(* IEC 61131-3 sources: plc-agent/examples, 6 files *)

(* ---- invalid.st ---- *)
PROGRAM Main
VAR_OUTPUT
    Motor : BOOL;
END_VAR

Motor := ;
END_PROGRAM

(* ---- minimal.st ---- *)
PROGRAM Main
VAR_INPUT
    Start : BOOL;
END_VAR
VAR_OUTPUT
    Motor : BOOL;
END_VAR

Motor := Start;
END_PROGRAM

(* ---- motor_start_stop.st ---- *)
PROGRAM Main
VAR
    Start AT %IX0.0 : BOOL;
    Stop AT %IX0.1 : BOOL;
    Motor AT %QX0.0 : BOOL;
END_VAR
VAR
    StartEdge : R_TRIG;
    RunTimer : TON;
    Running : BOOL := FALSE;
END_VAR

StartEdge(CLK := Start);
IF Stop THEN
    Running := FALSE;
ELSIF StartEdge.Q AND NOT Running THEN
    Running := TRUE;
END_IF;

RunTimer(IN := Running, PT := T#10s);
IF RunTimer.Q THEN
    Running := FALSE;
END_IF;
Motor := Running;
END_PROGRAM

CONFIGURATION Config0
    RESOURCE Res0 ON PLC
        TASK MainTask(INTERVAL := T#20ms, PRIORITY := 0);
        PROGRAM Inst0 WITH MainTask : Main;
    END_RESOURCE
END_CONFIGURATION

(* ---- p2_delay_10s.st ---- *)
PROGRAM Main
VAR
    Start AT %IX0.0 : BOOL;
    Motor AT %QX0.0 : BOOL;
END_VAR
VAR
    Timer1 : TON;
END_VAR

Timer1(IN := Start, PT := T#10s);
Motor := Timer1.Q;
END_PROGRAM

CONFIGURATION Config0
    RESOURCE Res0 ON PLC
        TASK MainTask(INTERVAL := T#20ms, PRIORITY := 0);
        PROGRAM Inst0 WITH MainTask : Main;
    END_RESOURCE
END_CONFIGURATION

(* ---- problem_001_solution.st ---- *)
PROGRAM Main
VAR
    Start AT %IX0.0 : BOOL;
    Stop AT %IX0.1 : BOOL;
    Motor AT %QX0.0 : BOOL;
END_VAR

Motor := Start AND NOT Stop;
END_PROGRAM

CONFIGURATION Config0
    RESOURCE Res0 ON PLC
        TASK MainTask(INTERVAL := T#20ms, PRIORITY := 0);
        PROGRAM Inst0 WITH MainTask : Main;
    END_RESOURCE
END_CONFIGURATION

(* ---- runtime_minimal.st ---- *)
PROGRAM Main
VAR
    Heartbeat AT %QX0.0 : BOOL;
END_VAR

Heartbeat := NOT Heartbeat;
END_PROGRAM

CONFIGURATION Config0
    RESOURCE Res0 ON PLC
        TASK MainTask(INTERVAL := T#100ms, PRIORITY := 0);
        PROGRAM Inst0 WITH MainTask : Main;
    END_RESOURCE
END_CONFIGURATION
